// Conveyor control interface — extends I_StateMachine
INTERFACE I_Conveyor EXTENDS I_StateMachine

METHOD Start : BOOL
VAR_INPUT
    fSpeed : LREAL; // Belt speed [m/s], 0 = use nominal
END_VAR
END_METHOD

METHOD Stop : BOOL
VAR_INPUT
END_VAR
END_METHOD

METHOD SetSpeed : BOOL
VAR_INPUT
    fSpeed : LREAL;
END_VAR
END_METHOD

METHOD IsRunning : BOOL
VAR_INPUT
END_VAR
END_METHOD

METHOD IsBlocked : BOOL
VAR_INPUT
END_VAR
END_METHOD

METHOD ProductPresent : BOOL
VAR_INPUT
END_VAR
END_METHOD

END_INTERFACE

(* stored: Version 1.1.0.1, ProductVersion 3.1.4024.12
   Itf I_Conveyor: Id {E4046036-9261-4C64-BEDC-CC645B10D032}
   Method Start: Id {1D89C373-DDDC-4D17-AB1E-FAC20BBD7008}
   Method Stop: Id {B456A3D0-11A4-4C26-A41C-01D54898B4DE}
   Method SetSpeed: Id {389E1B63-631C-43A5-90B8-E7D833BD1D97}
   Method IsRunning: Id {6D7A5652-B442-4F3C-BB61-DF49BC684A3D}
   Method IsBlocked: Id {85E469D6-117C-43DC-A95B-33B38EE99F3D}
   Method ProductPresent: Id {3F471449-B745-4E2C-93BC-5FC91285654C} *)
